// Mitsubishi GX Works2 project: 清洗机下线11.1修改   PLC: Q03UDE

PROGRAM INITIALI
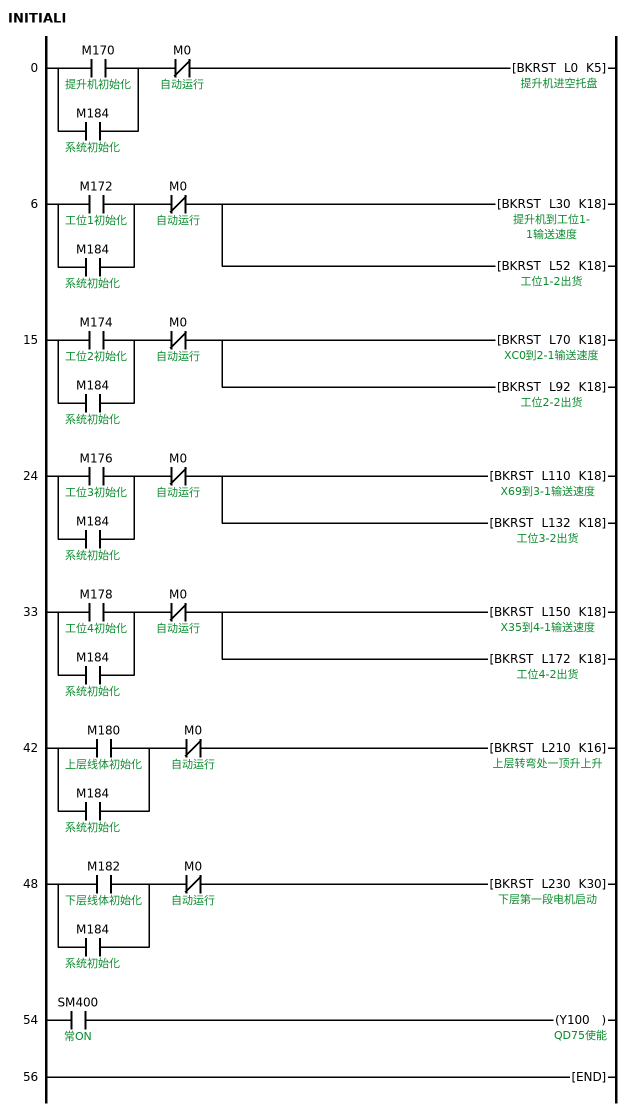
0     LD      M170  ; 提升机初始化
      OR      M184  ; 系统初始化
      ANI     M0  ; 自动运行
      BKRST   L0 K5  ; 提升机进空托盘
6     LD      M172  ; 工位1初始化
      OR      M184  ; 系统初始化
      ANI     M0  ; 自动运行
      BKRST   L30 K18  ; 提升机到工位1-1输送速度
      BKRST   L52 K18  ; 工位1-2出货
15    LD      M174  ; 工位2初始化
      OR      M184  ; 系统初始化
      ANI     M0  ; 自动运行
      BKRST   L70 K18  ; XC0到2-1输送速度
      BKRST   L92 K18  ; 工位2-2出货
24    LD      M176  ; 工位3初始化
      OR      M184  ; 系统初始化
      ANI     M0  ; 自动运行
      BKRST   L110 K18  ; X69到3-1输送速度
      BKRST   L132 K18  ; 工位3-2出货
33    LD      M178  ; 工位4初始化
      OR      M184  ; 系统初始化
      ANI     M0  ; 自动运行
      BKRST   L150 K18  ; X35到4-1输送速度
      BKRST   L172 K18  ; 工位4-2出货
42    LD      M180  ; 上层线体初始化
      OR      M184  ; 系统初始化
      ANI     M0  ; 自动运行
      BKRST   L210 K16  ; 上层转弯处一顶升上升
48    LD      M182  ; 下层线体初始化
      OR      M184  ; 系统初始化
      ANI     M0  ; 自动运行
      BKRST   L230 K30  ; 下层第一段电机启动
54    LD      SM400  ; 常ON
      OUT     Y100  ; QD75使能
56    END
END_PROGRAM

PROGRAM ALARM
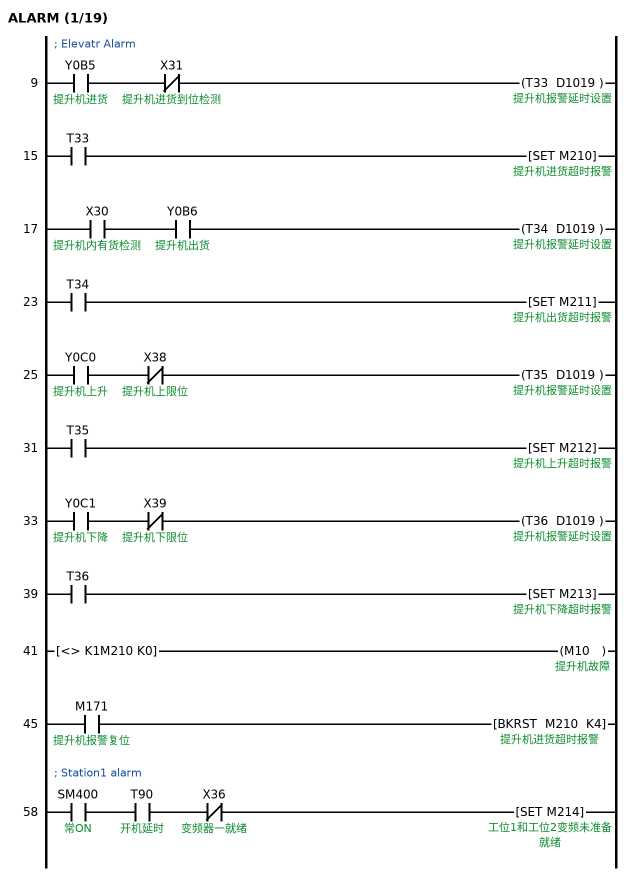
; Elevatr Alarm
9     LD      Y0B5  ; 提升机进货
      ANI     X31  ; 提升机进货到位检测
      OUT     T33 D1019  ; 提升机报警延时设置
15    LD      T33
      SET     M210  ; 提升机进货超时报警
17    LD      X30  ; 提升机内有货检测
      AND     Y0B6  ; 提升机出货
      OUT     T34 D1019  ; 提升机报警延时设置
23    LD      T34
      SET     M211  ; 提升机出货超时报警
25    LD      Y0C0  ; 提升机上升
      ANI     X38  ; 提升机上限位
      OUT     T35 D1019  ; 提升机报警延时设置
31    LD      T35
      SET     M212  ; 提升机上升超时报警
33    LD      Y0C1  ; 提升机下降
      ANI     X39  ; 提升机下限位
      OUT     T36 D1019  ; 提升机报警延时设置
39    LD      T36
      SET     M213  ; 提升机下降超时报警
41    LD<>    K1M210 K0  ; 提升机进货超时报警
      OUT     M10  ; 提升机故障
45    LD      M171  ; 提升机报警复位
      BKRST   M210 K4
; Station1 alarm
58    LD      SM400  ; 常ON
      AND     T90  ; 开机延时
      ANI     X36  ; 变频器一就绪
      SET     M214  ; 工位1和工位2变频未准备就绪
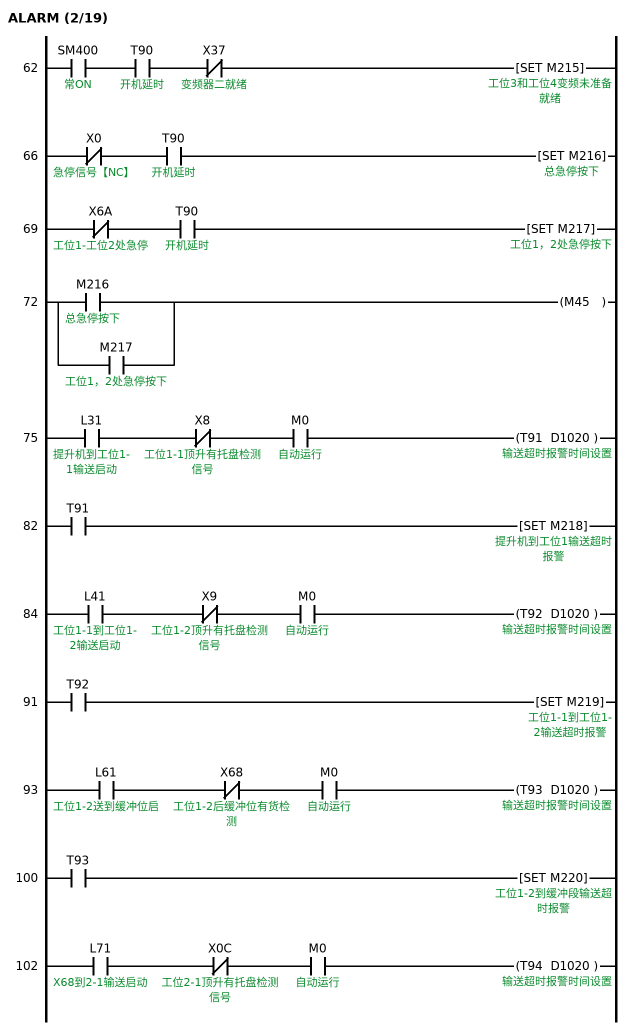
62    LD      SM400  ; 常ON
      AND     T90  ; 开机延时
      ANI     X37  ; 变频器二就绪
      SET     M215  ; 工位3和工位4变频未准备就绪
66    LDI     X0  ; 急停信号【NC】
      AND     T90  ; 开机延时
      SET     M216  ; 总急停按下
69    LDI     X6A  ; 工位1-工位2处急停
      AND     T90  ; 开机延时
      SET     M217  ; 工位1，2处急停按下
72    LD      M216  ; 总急停按下
      OR      M217  ; 工位1，2处急停按下
      OUT     M45
75    LD      L31  ; 提升机到工位1-1输送启动
      ANI     X8  ; 工位1-1顶升有托盘检测信号
      AND     M0  ; 自动运行
      OUT     T91 D1020  ; 输送超时报警时间设置
82    LD      T91
      SET     M218  ; 提升机到工位1输送超时报警
84    LD      L41  ; 工位1-1到工位1-2输送启动
      ANI     X9  ; 工位1-2顶升有托盘检测信号
      AND     M0  ; 自动运行
      OUT     T92 D1020  ; 输送超时报警时间设置
91    LD      T92
      SET     M219  ; 工位1-1到工位1-2输送超时报警
93    LD      L61  ; 工位1-2送到缓冲位启
      ANI     X68  ; 工位1-2后缓冲位有货检测
      AND     M0  ; 自动运行
      OUT     T93 D1020  ; 输送超时报警时间设置
100   LD      T93
      SET     M220  ; 工位1-2到缓冲段输送超时报警
102   LD      L71  ; X68到2-1输送启动
      ANI     X0C  ; 工位2-1顶升有托盘检测信号
      AND     M0  ; 自动运行
      OUT     T94 D1020  ; 输送超时报警时间设置
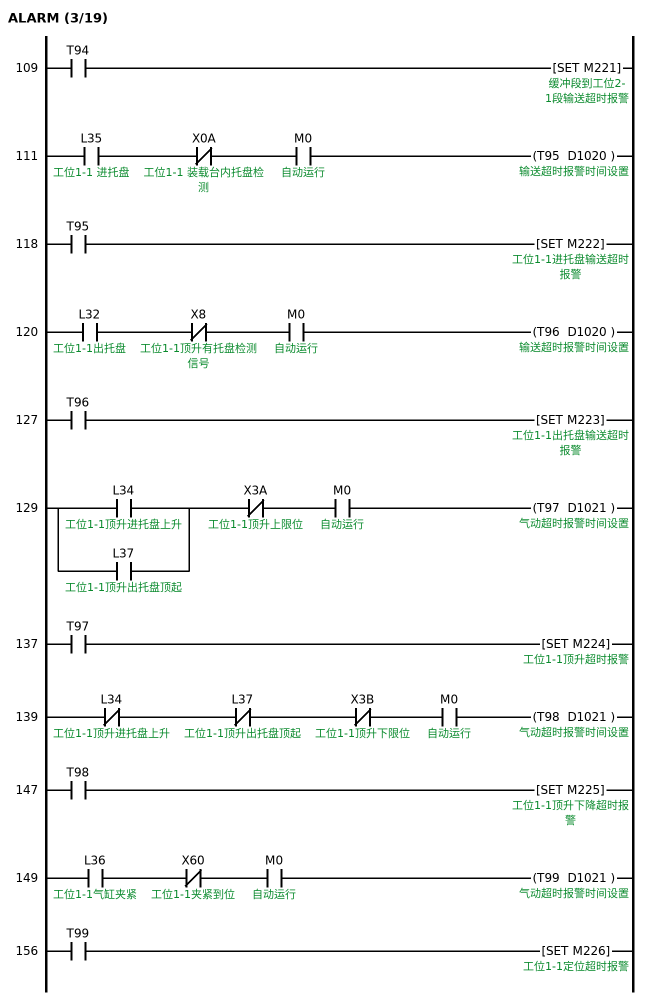
109   LD      T94
      SET     M221  ; 缓冲段到工位2-1段输送超时报警
111   LD      L35  ; 工位1-1 进托盘
      ANI     X0A  ; 工位1-1 装载台内托盘检测
      AND     M0  ; 自动运行
      OUT     T95 D1020  ; 输送超时报警时间设置
118   LD      T95
      SET     M222  ; 工位1-1进托盘输送超时报警
120   LD      L32  ; 工位1-1出托盘
      ANI     X8  ; 工位1-1顶升有托盘检测信号
      AND     M0  ; 自动运行
      OUT     T96 D1020  ; 输送超时报警时间设置
127   LD      T96
      SET     M223  ; 工位1-1出托盘输送超时报警
129   LD      L34  ; 工位1-1顶升进托盘上升
      OR      L37  ; 工位1-1顶升出托盘顶起
      ANI     X3A  ; 工位1-1顶升上限位
      AND     M0  ; 自动运行
      OUT     T97 D1021  ; 气动超时报警时间设置
137   LD      T97
      SET     M224  ; 工位1-1顶升超时报警
139   LDI     L34  ; 工位1-1顶升进托盘上升
      ANI     L37  ; 工位1-1顶升出托盘顶起
      ANI     X3B  ; 工位1-1顶升下限位
      AND     M0  ; 自动运行
      OUT     T98 D1021  ; 气动超时报警时间设置
147   LD      T98
      SET     M225  ; 工位1-1顶升下降超时报警
149   LD      L36  ; 工位1-1气缸夹紧
      ANI     X60  ; 工位1-1夹紧到位
      AND     M0  ; 自动运行
      OUT     T99 D1021  ; 气动超时报警时间设置
156   LD      T99
      SET     M226  ; 工位1-1定位超时报警
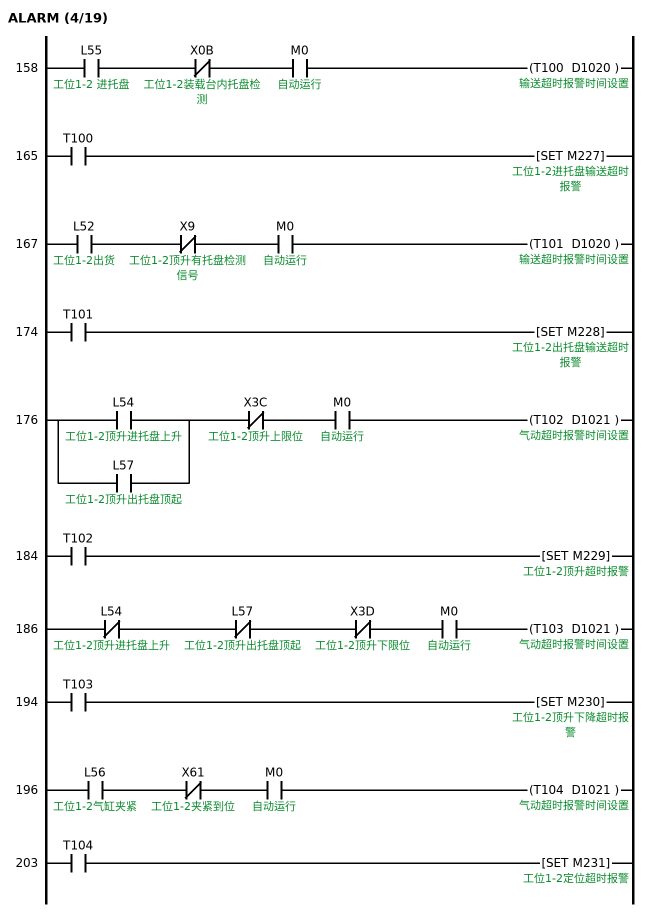
158   LD      L55  ; 工位1-2 进托盘
      ANI     X0B  ; 工位1-2装载台内托盘检测
      AND     M0  ; 自动运行
      OUT     T100 D1020  ; 输送超时报警时间设置
165   LD      T100
      SET     M227  ; 工位1-2进托盘输送超时报警
167   LD      L52  ; 工位1-2出货
      ANI     X9  ; 工位1-2顶升有托盘检测信号
      AND     M0  ; 自动运行
      OUT     T101 D1020  ; 输送超时报警时间设置
174   LD      T101
      SET     M228  ; 工位1-2出托盘输送超时报警
176   LD      L54  ; 工位1-2顶升进托盘上升
      OR      L57  ; 工位1-2顶升出托盘顶起
      ANI     X3C  ; 工位1-2顶升上限位
      AND     M0  ; 自动运行
      OUT     T102 D1021  ; 气动超时报警时间设置
184   LD      T102
      SET     M229  ; 工位1-2顶升超时报警
186   LDI     L54  ; 工位1-2顶升进托盘上升
      ANI     L57  ; 工位1-2顶升出托盘顶起
      ANI     X3D  ; 工位1-2顶升下限位
      AND     M0  ; 自动运行
      OUT     T103 D1021  ; 气动超时报警时间设置
194   LD      T103
      SET     M230  ; 工位1-2顶升下降超时报警
196   LD      L56  ; 工位1-2气缸夹紧
      ANI     X61  ; 工位1-2夹紧到位
      AND     M0  ; 自动运行
      OUT     T104 D1021  ; 气动超时报警时间设置
203   LD      T104
      SET     M231  ; 工位1-2定位超时报警
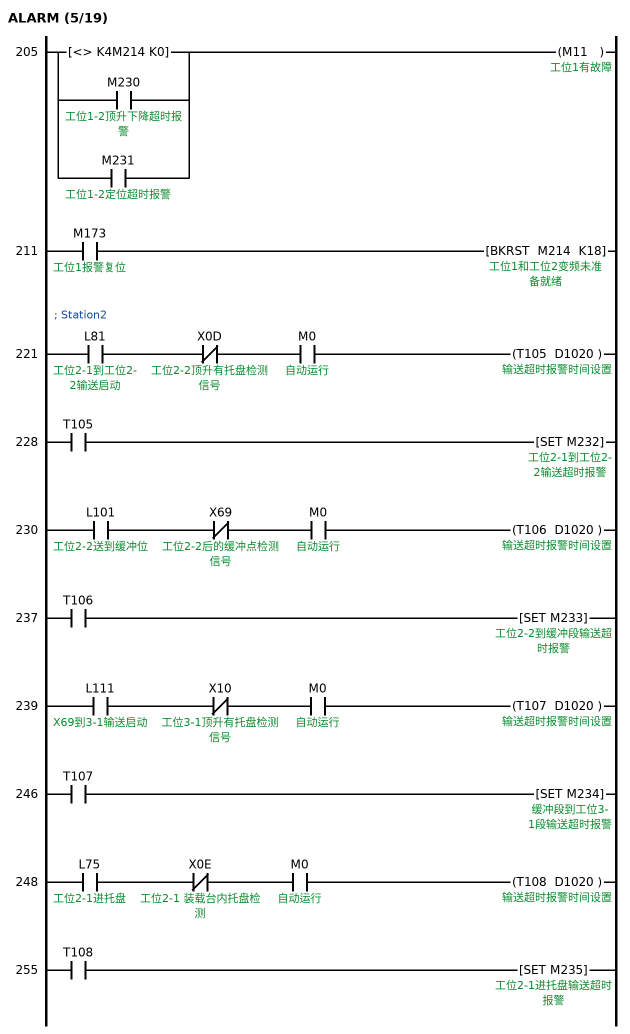
205   LD<>    K4M214 K0  ; 工位1和工位2变频未准备就绪
      OR      M230  ; 工位1-2顶升下降超时报警
      OR      M231  ; 工位1-2定位超时报警
      OUT     M11  ; 工位1有故障
211   LD      M173  ; 工位1报警复位
      BKRST   M214 K18
; Station2
221   LD      L81  ; 工位2-1到工位2-2输送启动
      ANI     X0D  ; 工位2-2顶升有托盘检测信号
      AND     M0  ; 自动运行
      OUT     T105 D1020  ; 输送超时报警时间设置
228   LD      T105
      SET     M232  ; 工位2-1到工位2-2输送超时报警
230   LD      L101  ; 工位2-2送到缓冲位
      ANI     X69  ; 工位2-2后的缓冲点检测信号
      AND     M0  ; 自动运行
      OUT     T106 D1020  ; 输送超时报警时间设置
237   LD      T106
      SET     M233  ; 工位2-2到缓冲段输送超时报警
239   LD      L111  ; X69到3-1输送启动
      ANI     X10  ; 工位3-1顶升有托盘检测信号
      AND     M0  ; 自动运行
      OUT     T107 D1020  ; 输送超时报警时间设置
246   LD      T107
      SET     M234  ; 缓冲段到工位3-1段输送超时报警
248   LD      L75  ; 工位2-1进托盘
      ANI     X0E  ; 工位2-1 装载台内托盘检测
      AND     M0  ; 自动运行
      OUT     T108 D1020  ; 输送超时报警时间设置
255   LD      T108
      SET     M235  ; 工位2-1进托盘输送超时报警
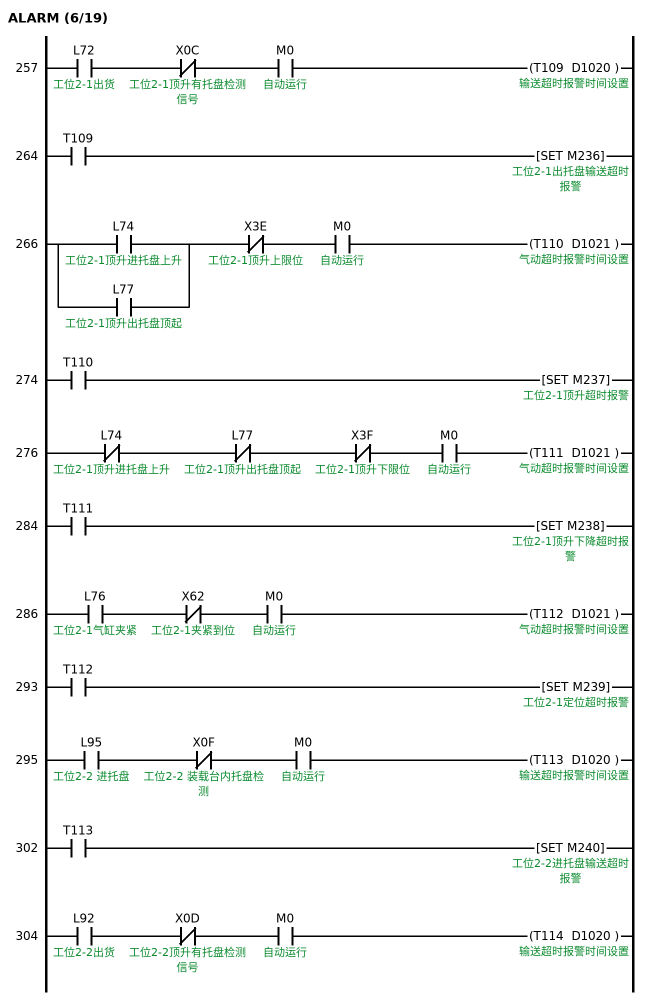
257   LD      L72  ; 工位2-1出货
      ANI     X0C  ; 工位2-1顶升有托盘检测信号
      AND     M0  ; 自动运行
      OUT     T109 D1020  ; 输送超时报警时间设置
264   LD      T109
      SET     M236  ; 工位2-1出托盘输送超时报警
266   LD      L74  ; 工位2-1顶升进托盘上升
      OR      L77  ; 工位2-1顶升出托盘顶起
      ANI     X3E  ; 工位2-1顶升上限位
      AND     M0  ; 自动运行
      OUT     T110 D1021  ; 气动超时报警时间设置
274   LD      T110
      SET     M237  ; 工位2-1顶升超时报警
276   LDI     L74  ; 工位2-1顶升进托盘上升
      ANI     L77  ; 工位2-1顶升出托盘顶起
      ANI     X3F  ; 工位2-1顶升下限位
      AND     M0  ; 自动运行
      OUT     T111 D1021  ; 气动超时报警时间设置
284   LD      T111
      SET     M238  ; 工位2-1顶升下降超时报警
286   LD      L76  ; 工位2-1气缸夹紧
      ANI     X62  ; 工位2-1夹紧到位
      AND     M0  ; 自动运行
      OUT     T112 D1021  ; 气动超时报警时间设置
293   LD      T112
      SET     M239  ; 工位2-1定位超时报警
295   LD      L95  ; 工位2-2 进托盘
      ANI     X0F  ; 工位2-2 装载台内托盘检测
      AND     M0  ; 自动运行
      OUT     T113 D1020  ; 输送超时报警时间设置
302   LD      T113
      SET     M240  ; 工位2-2进托盘输送超时报警
304   LD      L92  ; 工位2-2出货
      ANI     X0D  ; 工位2-2顶升有托盘检测信号
      AND     M0  ; 自动运行
      OUT     T114 D1020  ; 输送超时报警时间设置
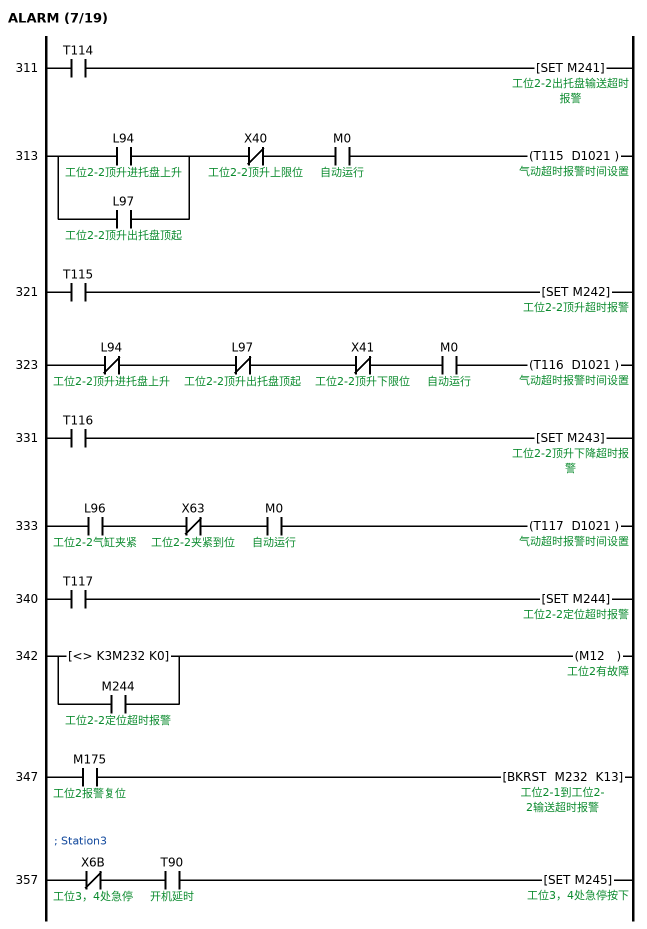
311   LD      T114
      SET     M241  ; 工位2-2出托盘输送超时报警
313   LD      L94  ; 工位2-2顶升进托盘上升
      OR      L97  ; 工位2-2顶升出托盘顶起
      ANI     X40  ; 工位2-2顶升上限位
      AND     M0  ; 自动运行
      OUT     T115 D1021  ; 气动超时报警时间设置
321   LD      T115
      SET     M242  ; 工位2-2顶升超时报警
323   LDI     L94  ; 工位2-2顶升进托盘上升
      ANI     L97  ; 工位2-2顶升出托盘顶起
      ANI     X41  ; 工位2-2顶升下限位
      AND     M0  ; 自动运行
      OUT     T116 D1021  ; 气动超时报警时间设置
331   LD      T116
      SET     M243  ; 工位2-2顶升下降超时报警
333   LD      L96  ; 工位2-2气缸夹紧
      ANI     X63  ; 工位2-2夹紧到位
      AND     M0  ; 自动运行
      OUT     T117 D1021  ; 气动超时报警时间设置
340   LD      T117
      SET     M244  ; 工位2-2定位超时报警
342   LD<>    K3M232 K0  ; 工位2-1到工位2-2输送超时报警
      OR      M244  ; 工位2-2定位超时报警
      OUT     M12  ; 工位2有故障
347   LD      M175  ; 工位2报警复位
      BKRST   M232 K13
; Station3
357   LDI     X6B  ; 工位3，4处急停
      AND     T90  ; 开机延时
      SET     M245  ; 工位3，4处急停按下
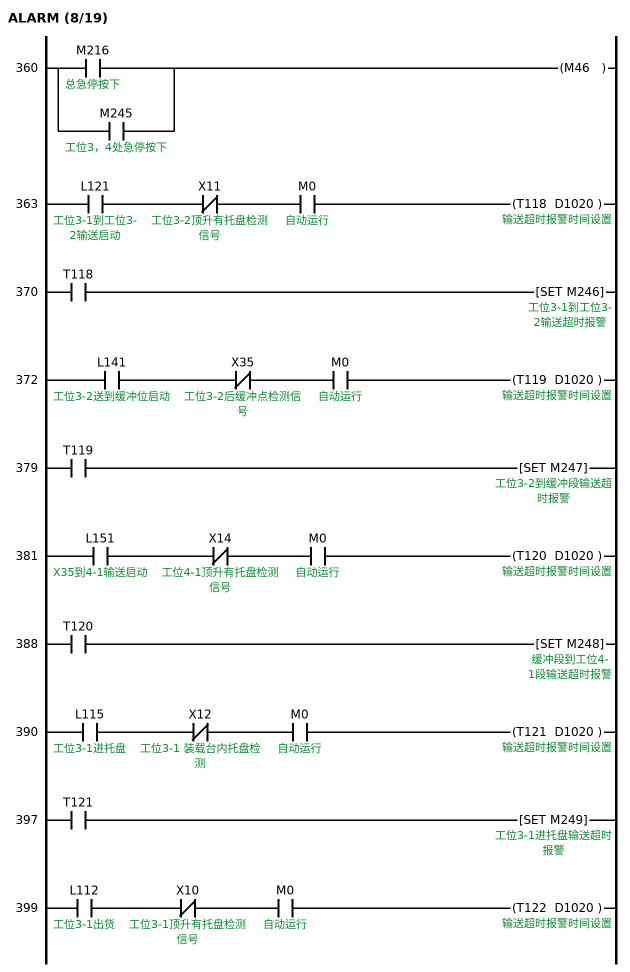
360   LD      M216  ; 总急停按下
      OR      M245  ; 工位3，4处急停按下
      OUT     M46
363   LD      L121  ; 工位3-1到工位3-2输送启动
      ANI     X11  ; 工位3-2顶升有托盘检测信号
      AND     M0  ; 自动运行
      OUT     T118 D1020  ; 输送超时报警时间设置
370   LD      T118
      SET     M246  ; 工位3-1到工位3-2输送超时报警
372   LD      L141  ; 工位3-2送到缓冲位启动
      ANI     X35  ; 工位3-2后缓冲点检测信号
      AND     M0  ; 自动运行
      OUT     T119 D1020  ; 输送超时报警时间设置
379   LD      T119
      SET     M247  ; 工位3-2到缓冲段输送超时报警
381   LD      L151  ; X35到4-1输送启动
      ANI     X14  ; 工位4-1顶升有托盘检测信号
      AND     M0  ; 自动运行
      OUT     T120 D1020  ; 输送超时报警时间设置
388   LD      T120
      SET     M248  ; 缓冲段到工位4-1段输送超时报警
390   LD      L115  ; 工位3-1进托盘
      ANI     X12  ; 工位3-1 装载台内托盘检测
      AND     M0  ; 自动运行
      OUT     T121 D1020  ; 输送超时报警时间设置
397   LD      T121
      SET     M249  ; 工位3-1进托盘输送超时报警
399   LD      L112  ; 工位3-1出货
      ANI     X10  ; 工位3-1顶升有托盘检测信号
      AND     M0  ; 自动运行
      OUT     T122 D1020  ; 输送超时报警时间设置
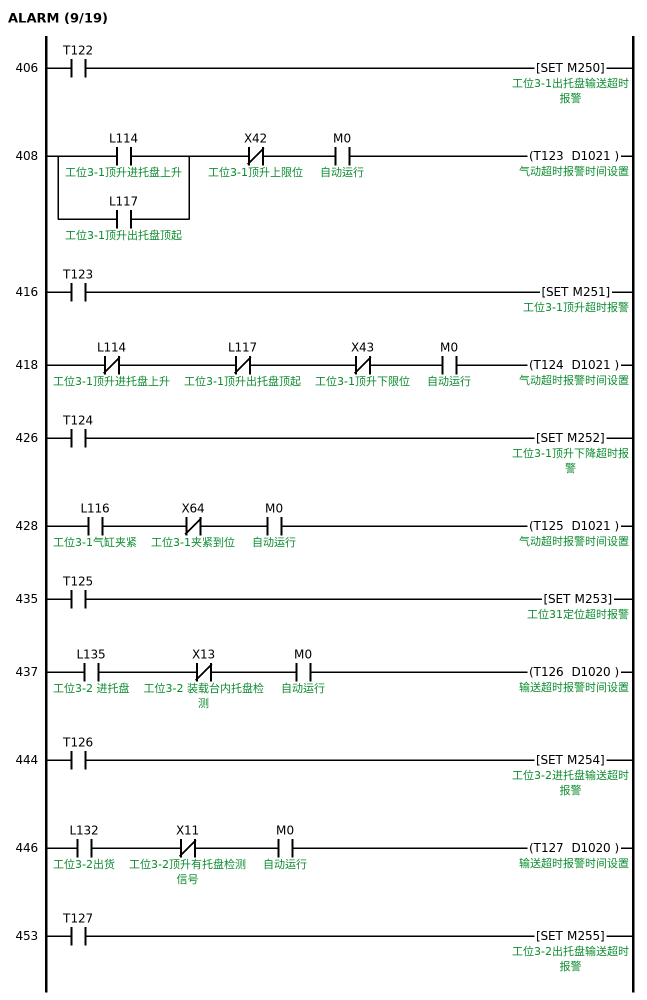
406   LD      T122
      SET     M250  ; 工位3-1出托盘输送超时报警
408   LD      L114  ; 工位3-1顶升进托盘上升
      OR      L117  ; 工位3-1顶升出托盘顶起
      ANI     X42  ; 工位3-1顶升上限位
      AND     M0  ; 自动运行
      OUT     T123 D1021  ; 气动超时报警时间设置
416   LD      T123
      SET     M251  ; 工位3-1顶升超时报警
418   LDI     L114  ; 工位3-1顶升进托盘上升
      ANI     L117  ; 工位3-1顶升出托盘顶起
      ANI     X43  ; 工位3-1顶升下限位
      AND     M0  ; 自动运行
      OUT     T124 D1021  ; 气动超时报警时间设置
426   LD      T124
      SET     M252  ; 工位3-1顶升下降超时报警
428   LD      L116  ; 工位3-1气缸夹紧
      ANI     X64  ; 工位3-1夹紧到位
      AND     M0  ; 自动运行
      OUT     T125 D1021  ; 气动超时报警时间设置
435   LD      T125
      SET     M253  ; 工位31定位超时报警
437   LD      L135  ; 工位3-2 进托盘
      ANI     X13  ; 工位3-2 装载台内托盘检测
      AND     M0  ; 自动运行
      OUT     T126 D1020  ; 输送超时报警时间设置
444   LD      T126
      SET     M254  ; 工位3-2进托盘输送超时报警
446   LD      L132  ; 工位3-2出货
      ANI     X11  ; 工位3-2顶升有托盘检测信号
      AND     M0  ; 自动运行
      OUT     T127 D1020  ; 输送超时报警时间设置
453   LD      T127
      SET     M255  ; 工位3-2出托盘输送超时报警
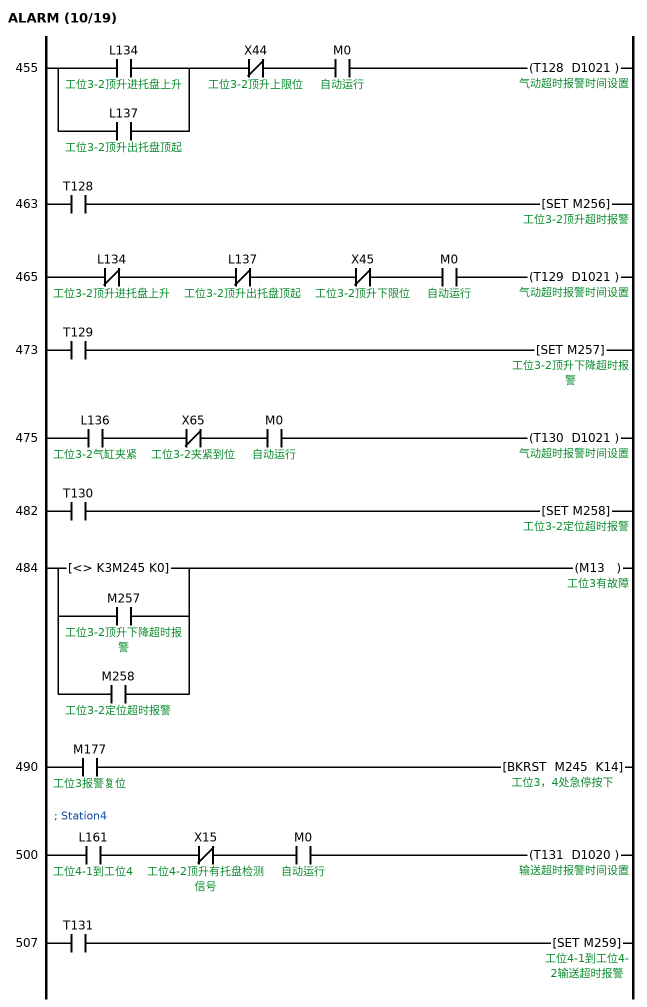
455   LD      L134  ; 工位3-2顶升进托盘上升
      OR      L137  ; 工位3-2顶升出托盘顶起
      ANI     X44  ; 工位3-2顶升上限位
      AND     M0  ; 自动运行
      OUT     T128 D1021  ; 气动超时报警时间设置
463   LD      T128
      SET     M256  ; 工位3-2顶升超时报警
465   LDI     L134  ; 工位3-2顶升进托盘上升
      ANI     L137  ; 工位3-2顶升出托盘顶起
      ANI     X45  ; 工位3-2顶升下限位
      AND     M0  ; 自动运行
      OUT     T129 D1021  ; 气动超时报警时间设置
473   LD      T129
      SET     M257  ; 工位3-2顶升下降超时报警
475   LD      L136  ; 工位3-2气缸夹紧
      ANI     X65  ; 工位3-2夹紧到位
      AND     M0  ; 自动运行
      OUT     T130 D1021  ; 气动超时报警时间设置
482   LD      T130
      SET     M258  ; 工位3-2定位超时报警
484   LD<>    K3M245 K0  ; 工位3，4处急停按下
      OR      M257  ; 工位3-2顶升下降超时报警
      OR      M258  ; 工位3-2定位超时报警
      OUT     M13  ; 工位3有故障
490   LD      M177  ; 工位3报警复位
      BKRST   M245 K14
; Station4
500   LD      L161  ; 工位4-1到工位4
      ANI     X15  ; 工位4-2顶升有托盘检测信号
      AND     M0  ; 自动运行
      OUT     T131 D1020  ; 输送超时报警时间设置
507   LD      T131
      SET     M259  ; 工位4-1到工位4-2输送超时报警
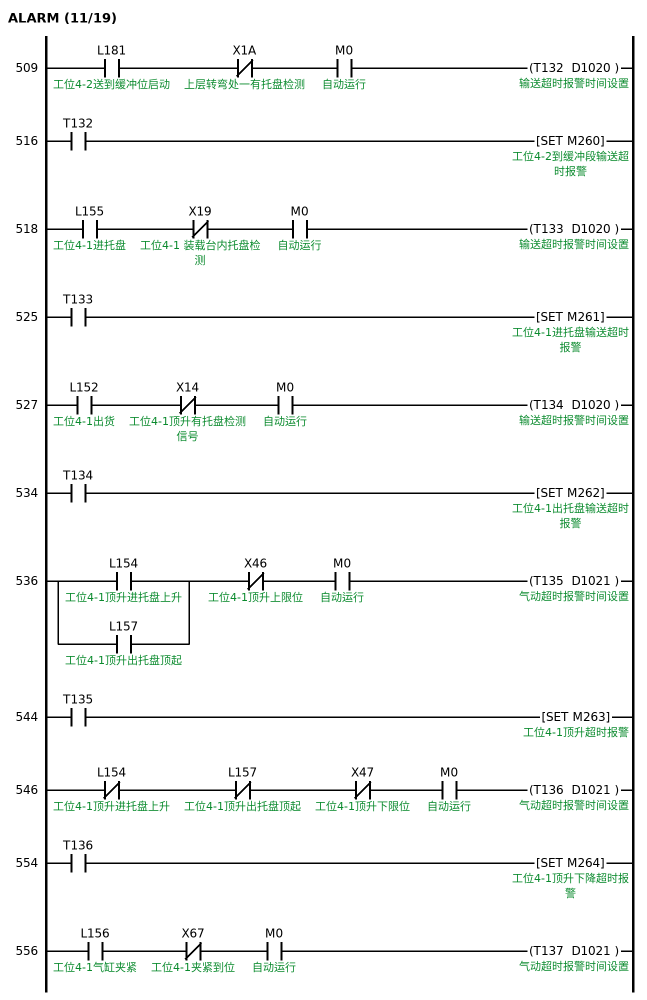
509   LD      L181  ; 工位4-2送到缓冲位启动
      ANI     X1A  ; 上层转弯处一有托盘检测
      AND     M0  ; 自动运行
      OUT     T132 D1020  ; 输送超时报警时间设置
516   LD      T132
      SET     M260  ; 工位4-2到缓冲段输送超时报警
518   LD      L155  ; 工位4-1进托盘
      ANI     X19  ; 工位4-1 装载台内托盘检测
      AND     M0  ; 自动运行
      OUT     T133 D1020  ; 输送超时报警时间设置
525   LD      T133
      SET     M261  ; 工位4-1进托盘输送超时报警
527   LD      L152  ; 工位4-1出货
      ANI     X14  ; 工位4-1顶升有托盘检测信号
      AND     M0  ; 自动运行
      OUT     T134 D1020  ; 输送超时报警时间设置
534   LD      T134
      SET     M262  ; 工位4-1出托盘输送超时报警
536   LD      L154  ; 工位4-1顶升进托盘上升
      OR      L157  ; 工位4-1顶升出托盘顶起
      ANI     X46  ; 工位4-1顶升上限位
      AND     M0  ; 自动运行
      OUT     T135 D1021  ; 气动超时报警时间设置
544   LD      T135
      SET     M263  ; 工位4-1顶升超时报警
546   LDI     L154  ; 工位4-1顶升进托盘上升
      ANI     L157  ; 工位4-1顶升出托盘顶起
      ANI     X47  ; 工位4-1顶升下限位
      AND     M0  ; 自动运行
      OUT     T136 D1021  ; 气动超时报警时间设置
554   LD      T136
      SET     M264  ; 工位4-1顶升下降超时报警
556   LD      L156  ; 工位4-1气缸夹紧
      ANI     X67  ; 工位4-1夹紧到位
      AND     M0  ; 自动运行
      OUT     T137 D1021  ; 气动超时报警时间设置
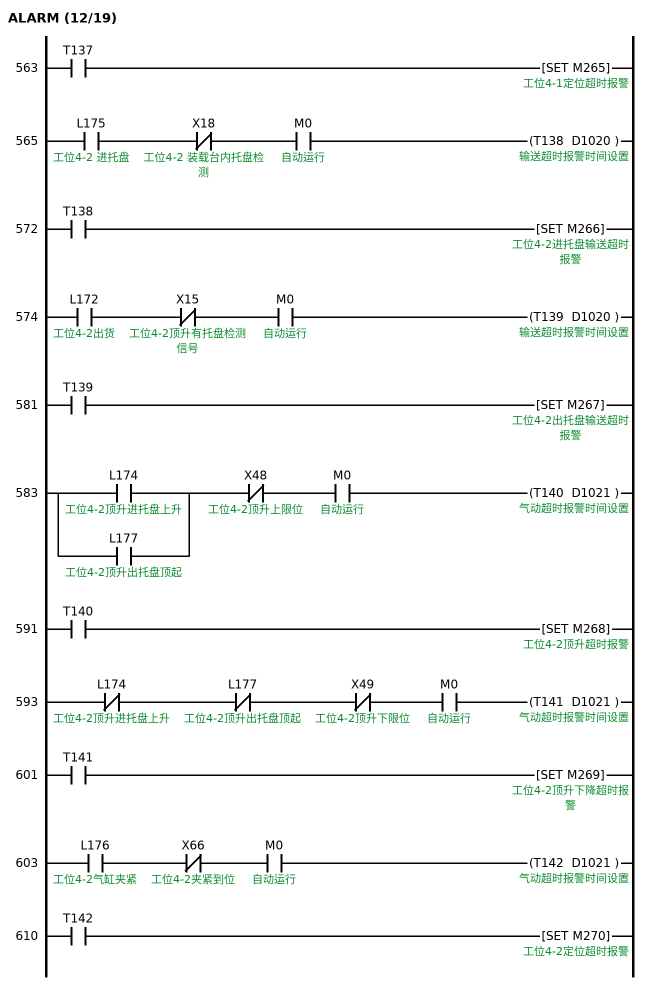
563   LD      T137
      SET     M265  ; 工位4-1定位超时报警
565   LD      L175  ; 工位4-2 进托盘
      ANI     X18  ; 工位4-2 装载台内托盘检测
      AND     M0  ; 自动运行
      OUT     T138 D1020  ; 输送超时报警时间设置
572   LD      T138
      SET     M266  ; 工位4-2进托盘输送超时报警
574   LD      L172  ; 工位4-2出货
      ANI     X15  ; 工位4-2顶升有托盘检测信号
      AND     M0  ; 自动运行
      OUT     T139 D1020  ; 输送超时报警时间设置
581   LD      T139
      SET     M267  ; 工位4-2出托盘输送超时报警
583   LD      L174  ; 工位4-2顶升进托盘上升
      OR      L177  ; 工位4-2顶升出托盘顶起
      ANI     X48  ; 工位4-2顶升上限位
      AND     M0  ; 自动运行
      OUT     T140 D1021  ; 气动超时报警时间设置
591   LD      T140
      SET     M268  ; 工位4-2顶升超时报警
593   LDI     L174  ; 工位4-2顶升进托盘上升
      ANI     L177  ; 工位4-2顶升出托盘顶起
      ANI     X49  ; 工位4-2顶升下限位
      AND     M0  ; 自动运行
      OUT     T141 D1021  ; 气动超时报警时间设置
601   LD      T141
      SET     M269  ; 工位4-2顶升下降超时报警
603   LD      L176  ; 工位4-2气缸夹紧
      ANI     X66  ; 工位4-2夹紧到位
      AND     M0  ; 自动运行
      OUT     T142 D1021  ; 气动超时报警时间设置
610   LD      T142
      SET     M270  ; 工位4-2定位超时报警
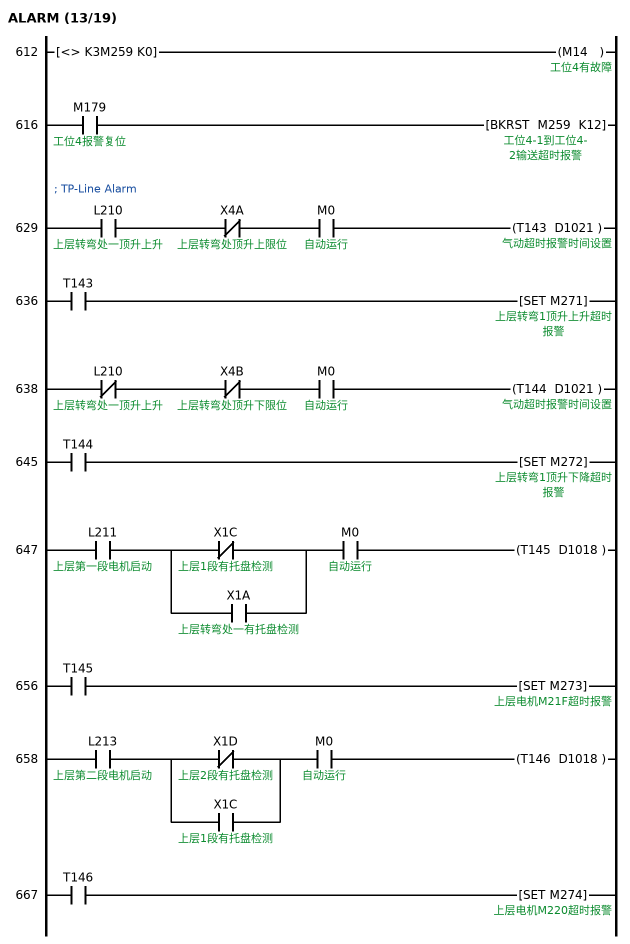
612   LD<>    K3M259 K0  ; 工位4-1到工位4-2输送超时报警
      OUT     M14  ; 工位4有故障
616   LD      M179  ; 工位4报警复位
      BKRST   M259 K12
; TP-Line Alarm
629   LD      L210  ; 上层转弯处一顶升上升
      ANI     X4A  ; 上层转弯处顶升上限位
      AND     M0  ; 自动运行
      OUT     T143 D1021  ; 气动超时报警时间设置
636   LD      T143
      SET     M271  ; 上层转弯1顶升上升超时报警
638   LDI     L210  ; 上层转弯处一顶升上升
      ANI     X4B  ; 上层转弯处顶升下限位
      AND     M0  ; 自动运行
      OUT     T144 D1021  ; 气动超时报警时间设置
645   LD      T144
      SET     M272  ; 上层转弯1顶升下降超时报警
647   LD      L211  ; 上层第一段电机启动
      LDI     X1C  ; 上层1段有托盘检测
      OR      X1A  ; 上层转弯处一有托盘检测
      ANB
      AND     M0  ; 自动运行
      OUT     T145 D1018
656   LD      T145
      SET     M273  ; 上层电机M21F超时报警
658   LD      L213  ; 上层第二段电机启动
      LDI     X1D  ; 上层2段有托盘检测
      OR      X1C  ; 上层1段有托盘检测
      ANB
      AND     M0  ; 自动运行
      OUT     T146 D1018
667   LD      T146
      SET     M274  ; 上层电机M220超时报警
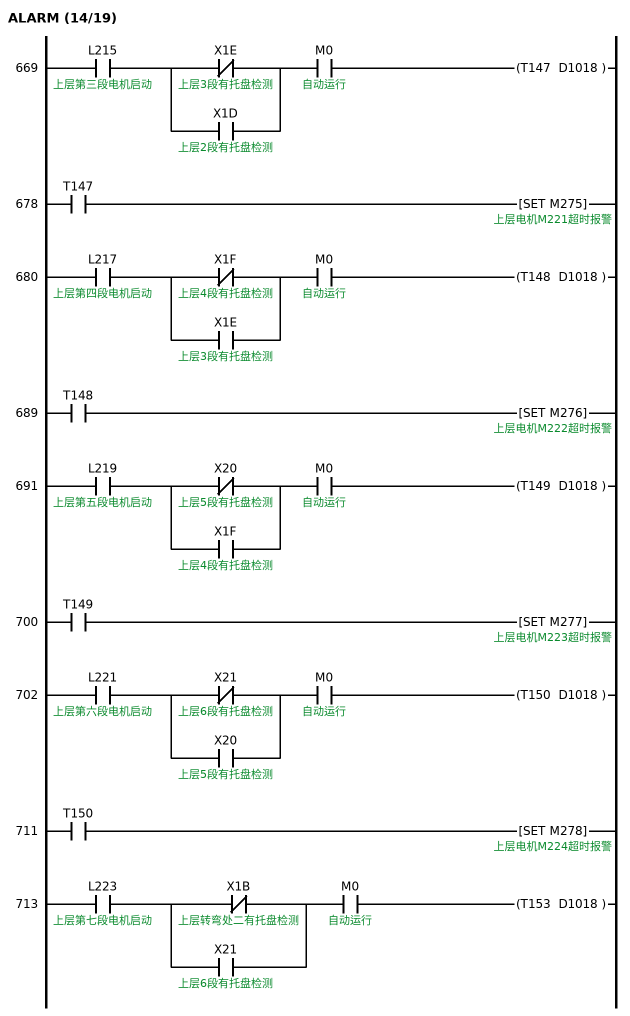
669   LD      L215  ; 上层第三段电机启动
      LDI     X1E  ; 上层3段有托盘检测
      OR      X1D  ; 上层2段有托盘检测
      ANB
      AND     M0  ; 自动运行
      OUT     T147 D1018
678   LD      T147
      SET     M275  ; 上层电机M221超时报警
680   LD      L217  ; 上层第四段电机启动
      LDI     X1F  ; 上层4段有托盘检测
      OR      X1E  ; 上层3段有托盘检测
      ANB
      AND     M0  ; 自动运行
      OUT     T148 D1018
689   LD      T148
      SET     M276  ; 上层电机M222超时报警
691   LD      L219  ; 上层第五段电机启动
      LDI     X20  ; 上层5段有托盘检测
      OR      X1F  ; 上层4段有托盘检测
      ANB
      AND     M0  ; 自动运行
      OUT     T149 D1018
700   LD      T149
      SET     M277  ; 上层电机M223超时报警
702   LD      L221  ; 上层第六段电机启动
      LDI     X21  ; 上层6段有托盘检测
      OR      X20  ; 上层5段有托盘检测
      ANB
      AND     M0  ; 自动运行
      OUT     T150 D1018
711   LD      T150
      SET     M278  ; 上层电机M224超时报警
713   LD      L223  ; 上层第七段电机启动
      LDI     X1B  ; 上层转弯处二有托盘检测
      OR      X21  ; 上层6段有托盘检测
      ANB
      AND     M0  ; 自动运行
      OUT     T153 D1018
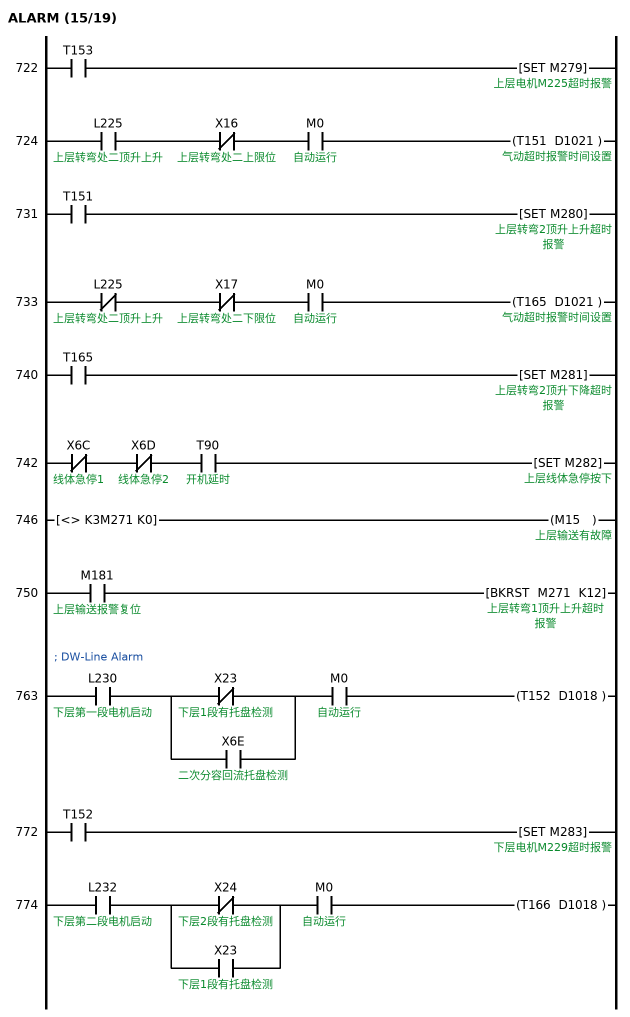
722   LD      T153
      SET     M279  ; 上层电机M225超时报警
724   LD      L225  ; 上层转弯处二顶升上升
      ANI     X16  ; 上层转弯处二上限位
      AND     M0  ; 自动运行
      OUT     T151 D1021  ; 气动超时报警时间设置
731   LD      T151
      SET     M280  ; 上层转弯2顶升上升超时报警
733   LDI     L225  ; 上层转弯处二顶升上升
      ANI     X17  ; 上层转弯处二下限位
      AND     M0  ; 自动运行
      OUT     T165 D1021  ; 气动超时报警时间设置
740   LD      T165
      SET     M281  ; 上层转弯2顶升下降超时报警
742   LDI     X6C  ; 线体急停1
      ANI     X6D  ; 线体急停2
      AND     T90  ; 开机延时
      SET     M282  ; 上层线体急停按下
746   LD<>    K3M271 K0  ; 上层转弯1顶升上升超时报警
      OUT     M15  ; 上层输送有故障
750   LD      M181  ; 上层输送报警复位
      BKRST   M271 K12
; DW-Line Alarm
763   LD      L230  ; 下层第一段电机启动
      LDI     X23  ; 下层1段有托盘检测
      OR      X6E  ; 二次分容回流托盘检测
      ANB
      AND     M0  ; 自动运行
      OUT     T152 D1018
772   LD      T152
      SET     M283  ; 下层电机M229超时报警
774   LD      L232  ; 下层第二段电机启动
      LDI     X24  ; 下层2段有托盘检测
      OR      X23  ; 下层1段有托盘检测
      ANB
      AND     M0  ; 自动运行
      OUT     T166 D1018
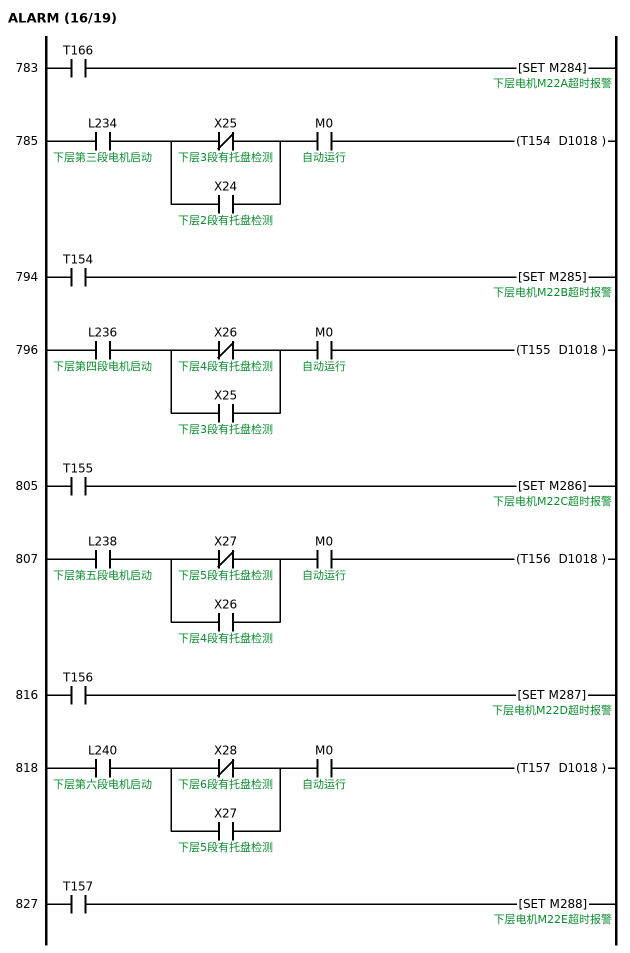
783   LD      T166
      SET     M284  ; 下层电机M22A超时报警
785   LD      L234  ; 下层第三段电机启动
      LDI     X25  ; 下层3段有托盘检测
      OR      X24  ; 下层2段有托盘检测
      ANB
      AND     M0  ; 自动运行
      OUT     T154 D1018
794   LD      T154
      SET     M285  ; 下层电机M22B超时报警
796   LD      L236  ; 下层第四段电机启动
      LDI     X26  ; 下层4段有托盘检测
      OR      X25  ; 下层3段有托盘检测
      ANB
      AND     M0  ; 自动运行
      OUT     T155 D1018
805   LD      T155
      SET     M286  ; 下层电机M22C超时报警
807   LD      L238  ; 下层第五段电机启动
      LDI     X27  ; 下层5段有托盘检测
      OR      X26  ; 下层4段有托盘检测
      ANB
      AND     M0  ; 自动运行
      OUT     T156 D1018
816   LD      T156
      SET     M287  ; 下层电机M22D超时报警
818   LD      L240  ; 下层第六段电机启动
      LDI     X28  ; 下层6段有托盘检测
      OR      X27  ; 下层5段有托盘检测
      ANB
      AND     M0  ; 自动运行
      OUT     T157 D1018
827   LD      T157
      SET     M288  ; 下层电机M22E超时报警
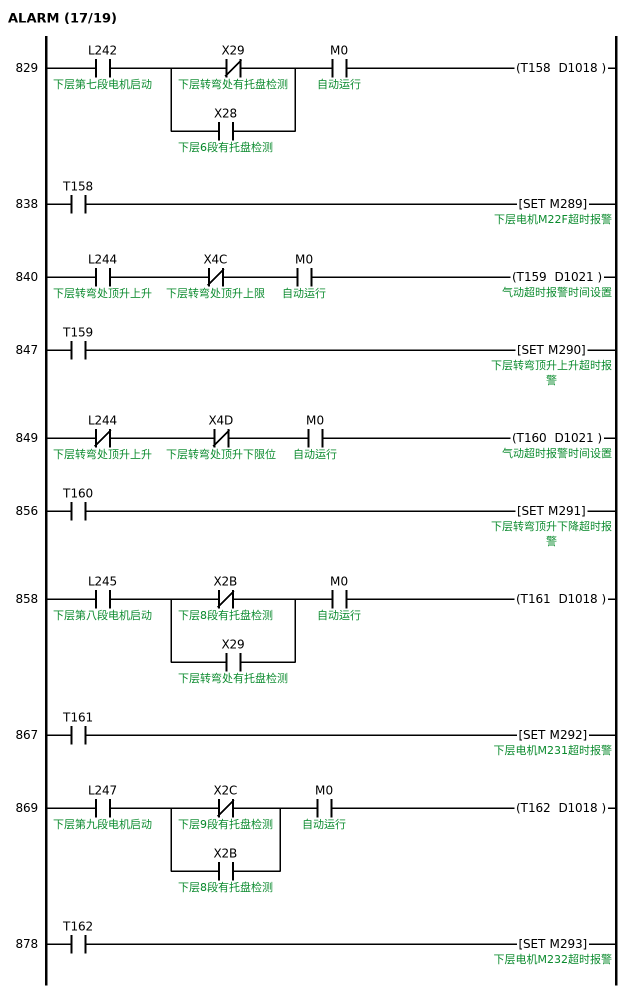
829   LD      L242  ; 下层第七段电机启动
      LDI     X29  ; 下层转弯处有托盘检测
      OR      X28  ; 下层6段有托盘检测
      ANB
      AND     M0  ; 自动运行
      OUT     T158 D1018
838   LD      T158
      SET     M289  ; 下层电机M22F超时报警
840   LD      L244  ; 下层转弯处顶升上升
      ANI     X4C  ; 下层转弯处顶升上限
      AND     M0  ; 自动运行
      OUT     T159 D1021  ; 气动超时报警时间设置
847   LD      T159
      SET     M290  ; 下层转弯顶升上升超时报警
849   LDI     L244  ; 下层转弯处顶升上升
      ANI     X4D  ; 下层转弯处顶升下限位
      AND     M0  ; 自动运行
      OUT     T160 D1021  ; 气动超时报警时间设置
856   LD      T160
      SET     M291  ; 下层转弯顶升下降超时报警
858   LD      L245  ; 下层第八段电机启动
      LDI     X2B  ; 下层8段有托盘检测
      OR      X29  ; 下层转弯处有托盘检测
      ANB
      AND     M0  ; 自动运行
      OUT     T161 D1018
867   LD      T161
      SET     M292  ; 下层电机M231超时报警
869   LD      L247  ; 下层第九段电机启动
      LDI     X2C  ; 下层9段有托盘检测
      OR      X2B  ; 下层8段有托盘检测
      ANB
      AND     M0  ; 自动运行
      OUT     T162 D1018
878   LD      T162
      SET     M293  ; 下层电机M232超时报警
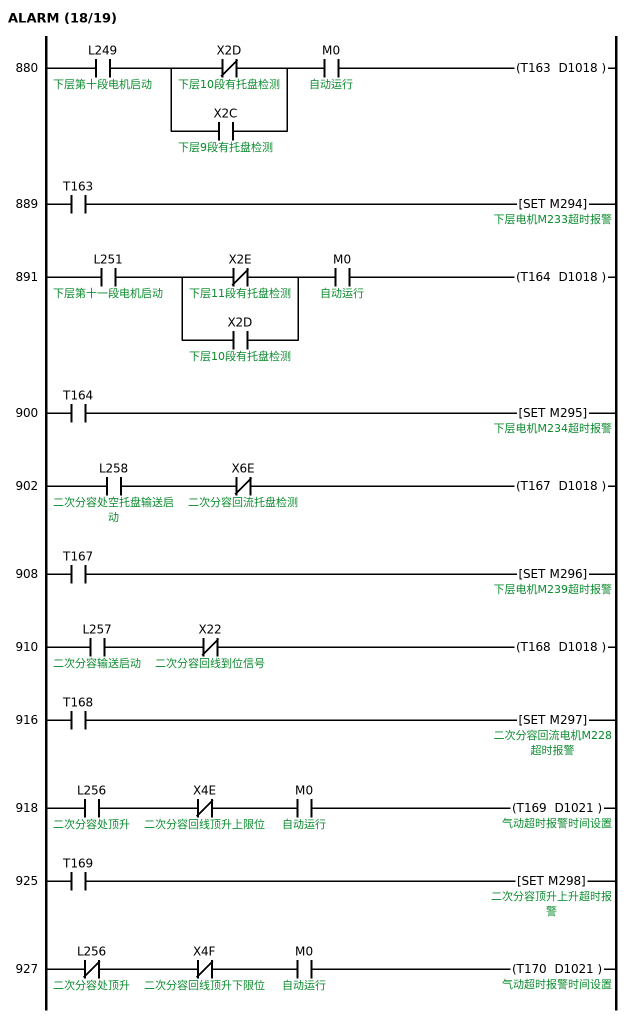
880   LD      L249  ; 下层第十段电机启动
      LDI     X2D  ; 下层10段有托盘检测
      OR      X2C  ; 下层9段有托盘检测
      ANB
      AND     M0  ; 自动运行
      OUT     T163 D1018
889   LD      T163
      SET     M294  ; 下层电机M233超时报警
891   LD      L251  ; 下层第十一段电机启动
      LDI     X2E  ; 下层11段有托盘检测
      OR      X2D  ; 下层10段有托盘检测
      ANB
      AND     M0  ; 自动运行
      OUT     T164 D1018
900   LD      T164
      SET     M295  ; 下层电机M234超时报警
902   LD      L258  ; 二次分容处空托盘输送启动
      ANI     X6E  ; 二次分容回流托盘检测
      OUT     T167 D1018
908   LD      T167
      SET     M296  ; 下层电机M239超时报警
910   LD      L257  ; 二次分容输送启动
      ANI     X22  ; 二次分容回线到位信号
      OUT     T168 D1018
916   LD      T168
      SET     M297  ; 二次分容回流电机M228超时报警
918   LD      L256  ; 二次分容处顶升
      ANI     X4E  ; 二次分容回线顶升上限位
      AND     M0  ; 自动运行
      OUT     T169 D1021  ; 气动超时报警时间设置
925   LD      T169
      SET     M298  ; 二次分容顶升上升超时报警
927   LDI     L256  ; 二次分容处顶升
      ANI     X4F  ; 二次分容回线顶升下限位
      AND     M0  ; 自动运行
      OUT     T170 D1021  ; 气动超时报警时间设置
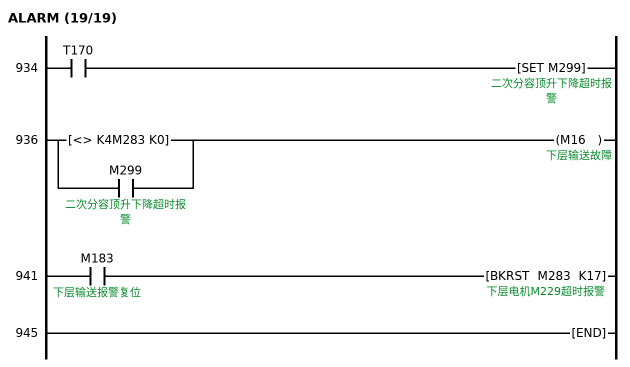
934   LD      T170
      SET     M299  ; 二次分容顶升下降超时报警
936   LD<>    K4M283 K0  ; 下层电机M229超时报警
      OR      M299  ; 二次分容顶升下降超时报警
      OUT     M16  ; 下层输送故障
941   LD      M183  ; 下层输送报警复位
      BKRST   M283 K17
945   END
END_PROGRAM

PROGRAM HMI
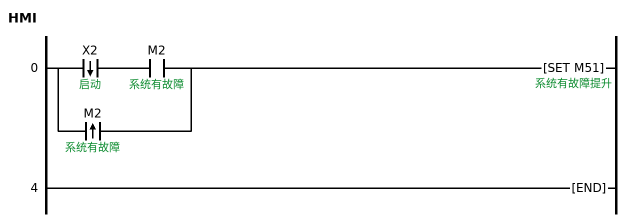
0     LDF     X2  ; 启动
      AND     M2  ; 系统有故障
      ORP     M2  ; 系统有故障
      SET     M51  ; 系统有故障提升
4     END
END_PROGRAM

PROGRAM ELEVATR
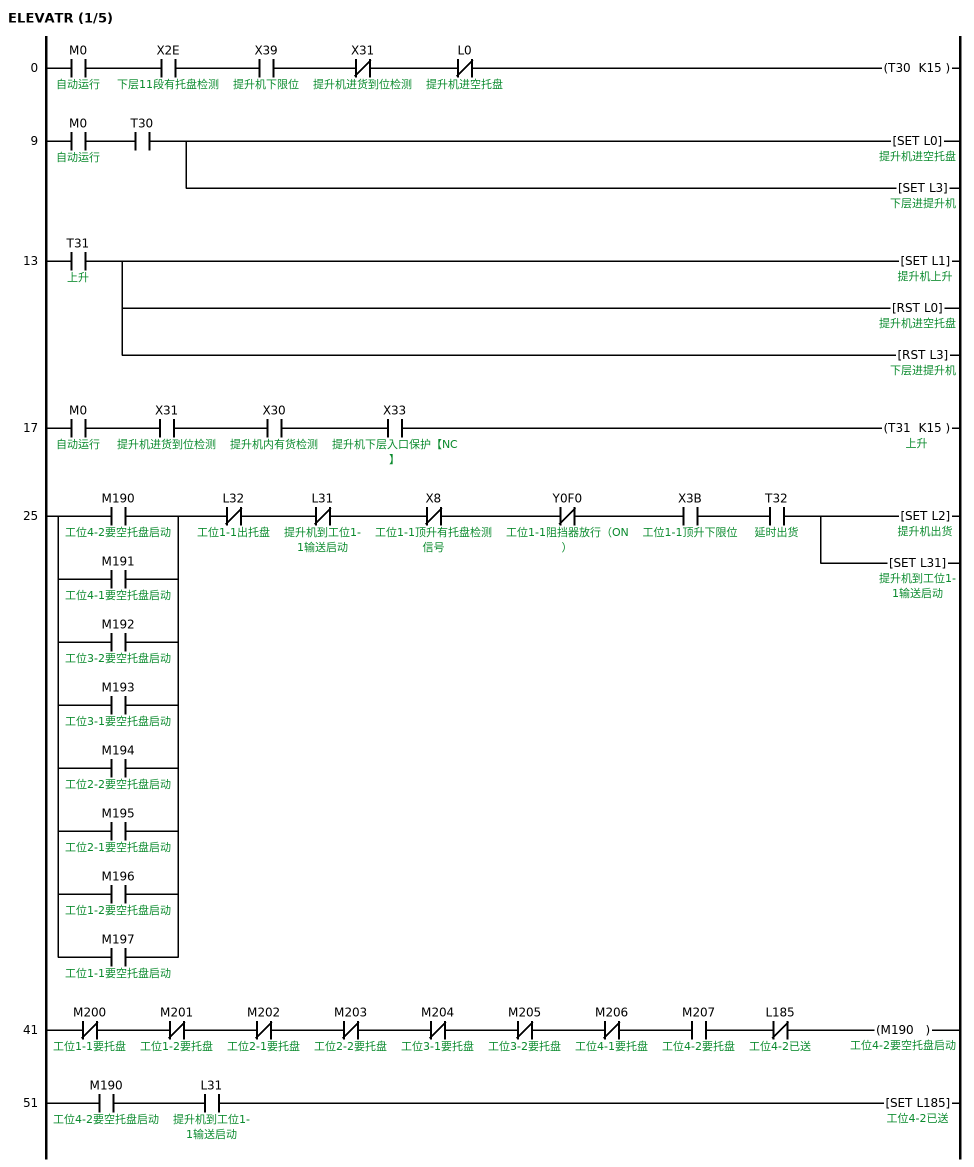
0     LD      M0  ; 自动运行
      AND     X2E  ; 下层11段有托盘检测
      AND     X39  ; 提升机下限位
      ANI     X31  ; 提升机进货到位检测
      ANI     L0  ; 提升机进空托盘
      OUT     T30 K15
9     LD      M0  ; 自动运行
      AND     T30
      SET     L0  ; 提升机进空托盘
      SET     L3  ; 下层进提升机
13    LD      T31  ; 上升
      SET     L1  ; 提升机上升
      RST     L0  ; 提升机进空托盘
      RST     L3  ; 下层进提升机
17    LD      M0  ; 自动运行
      AND     X31  ; 提升机进货到位检测
      AND     X30  ; 提升机内有货检测
      AND     X33  ; 提升机下层入口保护【NC】
      OUT     T31 K15  ; 上升
25    LD      M190  ; 工位4-2要空托盘启动
      OR      M191  ; 工位4-1要空托盘启动
      OR      M192  ; 工位3-2要空托盘启动
      OR      M193  ; 工位3-1要空托盘启动
      OR      M194  ; 工位2-2要空托盘启动
      OR      M195  ; 工位2-1要空托盘启动
      OR      M196  ; 工位1-2要空托盘启动
      OR      M197  ; 工位1-1要空托盘启动
      ANI     L32  ; 工位1-1出托盘
      ANI     L31  ; 提升机到工位1-1输送启动
      ANI     X8  ; 工位1-1顶升有托盘检测信号
      ANI     Y0F0  ; 工位1-1阻挡器放行（ON）
      AND     X3B  ; 工位1-1顶升下限位
      AND     T32  ; 延时出货
      SET     L2  ; 提升机出货
      SET     L31  ; 提升机到工位1-1输送启动
41    LDI     M200  ; 工位1-1要托盘
      ANI     M201  ; 工位1-2要托盘
      ANI     M202  ; 工位2-1要托盘
      ANI     M203  ; 工位2-2要托盘
      ANI     M204  ; 工位3-1要托盘
      ANI     M205  ; 工位3-2要托盘
      ANI     M206  ; 工位4-1要托盘
      AND     M207  ; 工位4-2要托盘
      ANI     L185  ; 工位4-2已送
      OUT     M190  ; 工位4-2要空托盘启动
51    LD      M190  ; 工位4-2要空托盘启动
      AND     L31  ; 提升机到工位1-1输送启动
      SET     L185  ; 工位4-2已送
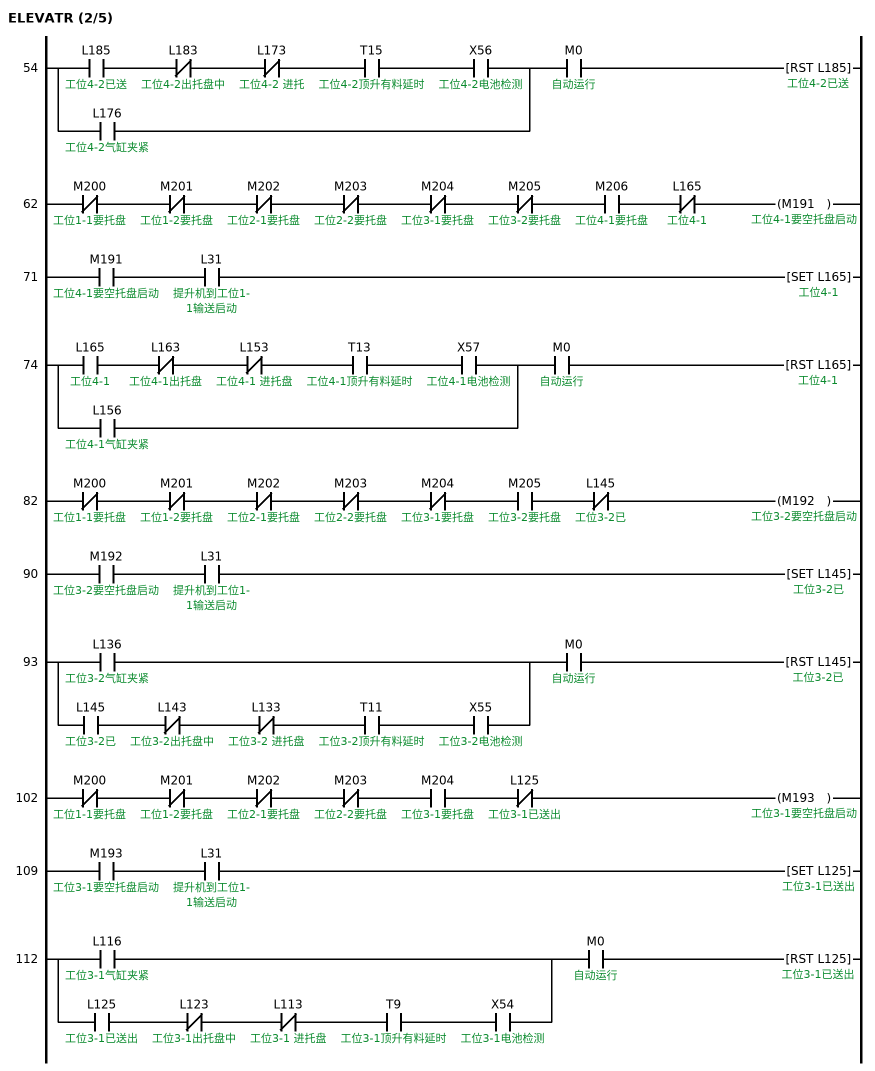
54    LD      L185  ; 工位4-2已送
      ANI     L183  ; 工位4-2出托盘中
      ANI     L173  ; 工位4-2 进托
      AND     T15  ; 工位4-2顶升有料延时
      AND     X56  ; 工位4-2电池检测
      OR      L176  ; 工位4-2气缸夹紧
      AND     M0  ; 自动运行
      RST     L185  ; 工位4-2已送
62    LDI     M200  ; 工位1-1要托盘
      ANI     M201  ; 工位1-2要托盘
      ANI     M202  ; 工位2-1要托盘
      ANI     M203  ; 工位2-2要托盘
      ANI     M204  ; 工位3-1要托盘
      ANI     M205  ; 工位3-2要托盘
      AND     M206  ; 工位4-1要托盘
      ANI     L165  ; 工位4-1
      OUT     M191  ; 工位4-1要空托盘启动
71    LD      M191  ; 工位4-1要空托盘启动
      AND     L31  ; 提升机到工位1-1输送启动
      SET     L165  ; 工位4-1
74    LD      L165  ; 工位4-1
      ANI     L163  ; 工位4-1出托盘
      ANI     L153  ; 工位4-1 进托盘
      AND     T13  ; 工位4-1顶升有料延时
      AND     X57  ; 工位4-1电池检测
      OR      L156  ; 工位4-1气缸夹紧
      AND     M0  ; 自动运行
      RST     L165  ; 工位4-1
82    LDI     M200  ; 工位1-1要托盘
      ANI     M201  ; 工位1-2要托盘
      ANI     M202  ; 工位2-1要托盘
      ANI     M203  ; 工位2-2要托盘
      ANI     M204  ; 工位3-1要托盘
      AND     M205  ; 工位3-2要托盘
      ANI     L145  ; 工位3-2已
      OUT     M192  ; 工位3-2要空托盘启动
90    LD      M192  ; 工位3-2要空托盘启动
      AND     L31  ; 提升机到工位1-1输送启动
      SET     L145  ; 工位3-2已
93    LD      L136  ; 工位3-2气缸夹紧
      LD      L145  ; 工位3-2已
      ANI     L143  ; 工位3-2出托盘中
      ANI     L133  ; 工位3-2 进托盘
      AND     T11  ; 工位3-2顶升有料延时
      AND     X55  ; 工位3-2电池检测
      ORB
      AND     M0  ; 自动运行
      RST     L145  ; 工位3-2已
102   LDI     M200  ; 工位1-1要托盘
      ANI     M201  ; 工位1-2要托盘
      ANI     M202  ; 工位2-1要托盘
      ANI     M203  ; 工位2-2要托盘
      AND     M204  ; 工位3-1要托盘
      ANI     L125  ; 工位3-1已送出
      OUT     M193  ; 工位3-1要空托盘启动
109   LD      M193  ; 工位3-1要空托盘启动
      AND     L31  ; 提升机到工位1-1输送启动
      SET     L125  ; 工位3-1已送出
112   LD      L116  ; 工位3-1气缸夹紧
      LD      L125  ; 工位3-1已送出
      ANI     L123  ; 工位3-1出托盘中
      ANI     L113  ; 工位3-1 进托盘
      AND     T9  ; 工位3-1顶升有料延时
      AND     X54  ; 工位3-1电池检测
      ORB
      AND     M0  ; 自动运行
      RST     L125  ; 工位3-1已送出
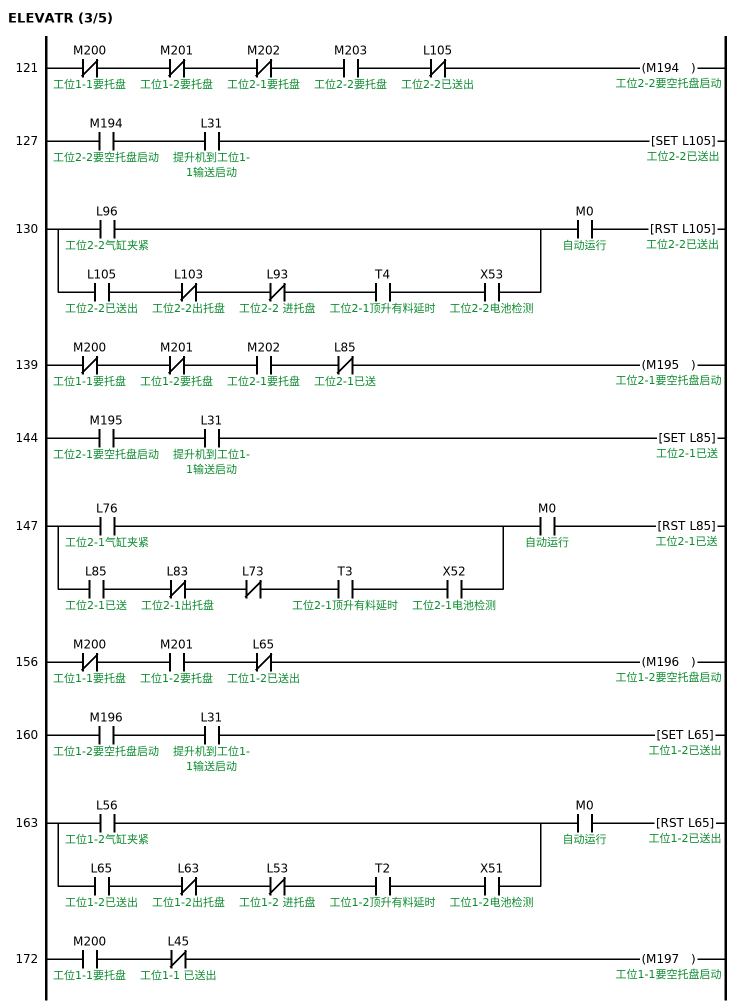
121   LDI     M200  ; 工位1-1要托盘
      ANI     M201  ; 工位1-2要托盘
      ANI     M202  ; 工位2-1要托盘
      AND     M203  ; 工位2-2要托盘
      ANI     L105  ; 工位2-2已送出
      OUT     M194  ; 工位2-2要空托盘启动
127   LD      M194  ; 工位2-2要空托盘启动
      AND     L31  ; 提升机到工位1-1输送启动
      SET     L105  ; 工位2-2已送出
130   LD      L96  ; 工位2-2气缸夹紧
      LD      L105  ; 工位2-2已送出
      ANI     L103  ; 工位2-2出托盘
      ANI     L93  ; 工位2-2 进托盘
      AND     T4  ; 工位2-1顶升有料延时
      AND     X53  ; 工位2-2电池检测
      ORB
      AND     M0  ; 自动运行
      RST     L105  ; 工位2-2已送出
139   LDI     M200  ; 工位1-1要托盘
      ANI     M201  ; 工位1-2要托盘
      AND     M202  ; 工位2-1要托盘
      ANI     L85  ; 工位2-1已送
      OUT     M195  ; 工位2-1要空托盘启动
144   LD      M195  ; 工位2-1要空托盘启动
      AND     L31  ; 提升机到工位1-1输送启动
      SET     L85  ; 工位2-1已送
147   LD      L76  ; 工位2-1气缸夹紧
      LD      L85  ; 工位2-1已送
      ANI     L83  ; 工位2-1出托盘
      ANI     L73
      AND     T3  ; 工位2-1顶升有料延时
      AND     X52  ; 工位2-1电池检测
      ORB
      AND     M0  ; 自动运行
      RST     L85  ; 工位2-1已送
156   LDI     M200  ; 工位1-1要托盘
      AND     M201  ; 工位1-2要托盘
      ANI     L65  ; 工位1-2已送出
      OUT     M196  ; 工位1-2要空托盘启动
160   LD      M196  ; 工位1-2要空托盘启动
      AND     L31  ; 提升机到工位1-1输送启动
      SET     L65  ; 工位1-2已送出
163   LD      L56  ; 工位1-2气缸夹紧
      LD      L65  ; 工位1-2已送出
      ANI     L63  ; 工位1-2出托盘
      ANI     L53  ; 工位1-2 进托盘
      AND     T2  ; 工位1-2顶升有料延时
      AND     X51  ; 工位1-2电池检测
      ORB
      AND     M0  ; 自动运行
      RST     L65  ; 工位1-2已送出
172   LD      M200  ; 工位1-1要托盘
      ANI     L45  ; 工位1-1 已送出
      OUT     M197  ; 工位1-1要空托盘启动
